ABB RAPID module: Module1.mod

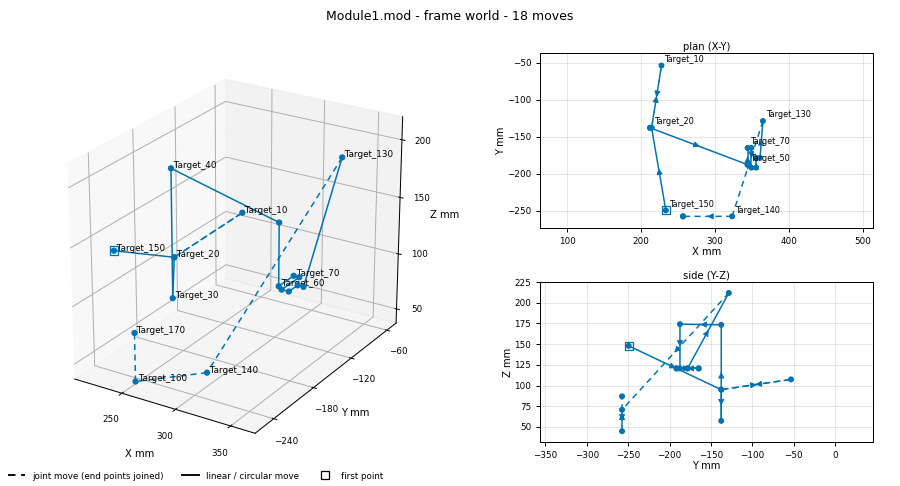
[picture p0: tool path of Module1.mod in frame world, 18 of 18 moves have a stored position in this frame; points joined in program order, loops and branches not executed]
MODULE Module1
	CONST robtarget Target_150:=[[233.211811557,-249.472208044,147.913605805],[0.066010562,-0.842421072,-0.111215201,-0.523068373],[0,0,1,4],[-101.964429524,9E+09,9E+09,9E+09,9E+09,9E+09]];
	CONST robtarget Target_20:=[[213.910672541,-137.748543138,95.059705176],[0.006071722,0.998222958,0.057306881,-0.015165169],[1,-2,2,4],[-108.944781509,9E+09,9E+09,9E+09,9E+09,9E+09]];
	CONST robtarget Target_10:=[[227.316998107,-53.532555281,107.421665526],[0.683227237,-0.728785964,0.024727998,-0.03821109],[1,-2,-1,5],[-167.584252868,9E+09,9E+09,9E+09,9E+09,9E+09]];
	CONST robtarget Target_30:=[[211.863267918,-137.748924149,57.377173818],[0.006071869,0.998222941,0.057307065,-0.015165513],[1,-2,2,4],[-109.556921499,9E+09,9E+09,9E+09,9E+09,9E+09]];
	CONST robtarget Target_40:=[[211.863400076,-137.749079805,173.323089952],[0.006071913,0.998222936,0.05730711,-0.015165653],[0,-2,2,4],[-107.511235642,9E+09,9E+09,9E+09,9E+09,9E+09]];
	CONST robtarget Target_50:=[[343.823237526,-187.587633041,174.130681723],[0.004947831,-0.734390317,-0.678530758,0.015568893],[1,-2,2,4],[-131.680598581,9E+09,9E+09,9E+09,9E+09,9E+09]];
	CONST robtarget Target_60:=[[343.823332743,-187.587817742,120.706896396],[0.004947883,-0.734390253,-0.678530825,0.015569024],[1,-2,1,4],[-131.680593152,9E+09,9E+09,9E+09,9E+09,9E+09]];
	CONST robtarget Target_70:=[[343.823447801,-164.995142165,120.706893277],[0.004947895,-0.734390281,-0.678530791,0.015569194],[1,-2,2,4],[-131.680593412,9E+09,9E+09,9E+09,9E+09,9E+09]];
	CONST robtarget Target_80:=[[348.888459482,-164.995370319,120.70680536],[0.004947855,-0.734390219,-0.678530854,0.015569383],[1,-2,2,4],[-131.680598828,9E+09,9E+09,9E+09,9E+09,9E+09]];
	CONST robtarget Target_90:=[[348.888540858,-191.668414254,120.706745959],[0.004947887,-0.734390121,-0.678530956,0.015569544],[1,-2,1,4],[-131.680598246,9E+09,9E+09,9E+09,9E+09,9E+09]];
	CONST robtarget Target_100:=[[355.358380618,-191.668647156,120.70674907],[0.004947865,-0.734390142,-0.67853093,0.015569706],[1,-2,1,4],[-131.680596176,9E+09,9E+09,9E+09,9E+09,9E+09]];
	CONST robtarget Target_110:=[[355.358457345,-178.436626801,120.70675146],[0.004947881,-0.734390135,-0.678530933,0.015569862],[1,-2,2,4],[-131.680595511,9E+09,9E+09,9E+09,9E+09,9E+09]];
	CONST robtarget Target_120:=[[360.613446573,-178.436857944,120.706640752],[0.004947923,-0.734390098,-0.678530968,0.01557007],[1,-2,1,4],[-131.680595457,9E+09,9E+09,9E+09,9E+09,9E+09]];
	CONST robtarget Target_130:=[[364.548930422,-128.598640756,211.83744596],[0.00494793,-0.734390022,-0.678531049,0.015570155],[1,-1,2,4],[-131.680594895,9E+09,9E+09,9E+09,9E+09,9E+09]];
	CONST robtarget Target_140:=[[322.811279064,-257.540101059,70.727887287],[0.004947975,-0.734389743,-0.678531327,0.015571183],[1,-2,1,4],[-131.680595261,9E+09,9E+09,9E+09,9E+09,9E+09]];
	CONST robtarget Target_160:=[[256.428591125,-257.540926286,44.886754917],[0.004948128,-0.734389716,-0.67853134,0.0155718],[1,-2,1,4],[-131.680599433,9E+09,9E+09,9E+09,9E+09,9E+09]];
	CONST robtarget Target_170:=[[256.428708938,-257.541118261,87.020832403],[0.004948122,-0.734389689,-0.678531366,0.01557197],[1,-2,1,4],[-131.680603505,9E+09,9E+09,9E+09,9E+09,9E+09]];
	PROC Path_10()
	    MoveJ Target_150,v1000,z100,Servo\WObj:=wobj0;
	    MoveL Target_20,v1000,z100,Servo\WObj:=wobj0;
	    MoveJ Target_10,v1000,z100,Servo\WObj:=wobj0;
	    WaitTime 2;
	    MoveJ Target_20,v1000,z100,Servo\WObj:=wobj0;
	    MoveL Target_30,v80,fine,Servo\WObj:=wobj0;
	    PulseDO attach_ring1;
	    WaitTime 1;
	    MoveL Target_40,v1000,z100,Servo\WObj:=wobj0;
	    MoveL Target_50,v1000,z100,Servo\WObj:=wobj0;
	    MoveL Target_60,v1000,z100,Servo\WObj:=wobj0;
	    MoveL Target_70,v1000,z100,Servo\WObj:=wobj0;
	    MoveL Target_80,v1000,z100,Servo\WObj:=wobj0;
	    MoveL Target_90,v1000,z100,Servo\WObj:=wobj0;
	    MoveL Target_100,v1000,z100,Servo\WObj:=wobj0;
	    MoveL Target_110,v1000,z100,Servo\WObj:=wobj0;
	    MoveL Target_120,v1000,z100,Servo\WObj:=wobj0;
	    MoveL Target_130,v1000,z100,Servo\WObj:=wobj0;
		MoveJ Target_140,v1000,z100,Servo\WObj:=wobj0;
		MoveJ Target_160,v1000,z100,Servo\WObj:=wobj0;
		WaitTime 5;
		PulseDO detach_ring1;
		WaitTime 2;
		MoveJ Target_170,v1000,z100,Servo\WObj:=wobj0;
	ENDPROC
	PROC main()
	    Path_10;
	ENDPROC
ENDMODULE
